// TIA Portal V19 export
FUNCTION "M_TolWindow" : Bool   // FC27, LAD
TITLE = CHECK IF ActPos is within tolerance window with Target
// stored: Access Published, SetENOAutomatically false
   VAR_INPUT
      ActPos : LReal;
      Target : LReal;
      PosWin : LReal;
      MODULE : LReal;
   END_VAR
   VAR_TEMP
      Pos : LReal;
      PosAbs : LReal;
   END_VAR
BEGIN

REGION Network 1: Delta with module
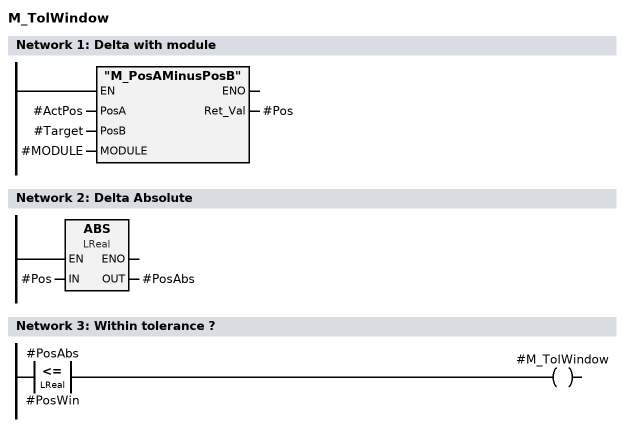
   RUNG wire#powerrail
      "M_PosAMinusPosB"(PosA := #ActPos, PosB := #Target, MODULE := #MODULE, Ret_Val => #Pos)
   END_RUNG
   // the same network as SCL:
   #Pos := "M_PosAMinusPosB"(PosA := #ActPos, PosB := #Target, MODULE := #MODULE);
END_REGION

REGION Network 2: Delta Absolute
   RUNG wire#powerrail
      { S7_Templates := "SrcType := LReal" } Abs(in := #Pos, out => #PosAbs)
   END_RUNG
   // the same network as SCL:
   #PosAbs := ABS(#Pos);
END_REGION

REGION Network 3: Within tolerance ?
   RUNG wire#powerrail
      { S7_Templates := "SrcType := LReal" } LE_Contact(in1 := #PosAbs, in2 := #PosWin)
      Coil( #M_TolWindow )
   END_RUNG
   // the same network as SCL:
   #M_TolWindow := #PosAbs <= #PosWin;
END_REGION
END_FUNCTION
